TEXTLIST CmdTxtList
  0 = 'INITIALISE'
  1 = 'AlarmReset'
  2 = 'ColumnAlarmReset'
  3 = 'TIUSlideIn'
  4 = 'TIUSlideOut'
  5 = 'TIUDrawerUp'
  6 = 'TIUDrawerDown'
  7 = 'TIUSlideOutRetry'
  8 = 'TIUSlideOutCancel'
  9 = 'DPSPowerON'
  10 = 'DPSPowerOFF'
  11 = 'DPSPowerAuto'
  12 = 'AP240ACPowerON'
  13 = 'AP240ACPowerOFF'
  14 = 'APAirValveON'
  15 = 'APAirValveOFF'
  16 = 'TstAirValveON'
  17 = 'TstAirValveOFF'
  18 = 'CellDoorOpen'
  19 = 'CellDoorClose'
  20 = 'CancelBuffer'
  21 = 'SetLEDON'
  22 = 'SetLEDOFF'
  23 = 'SetLEDBlink'
  24 = 'DCCellFrontDoorOpen'
  25 = 'DCCellFrontDoorClose'
  26 = 'TIUSocketAirOn_1'
  27 = 'TIUSocketAirOn_2'
  28 = 'TIUSocketAirOff_1'
  29 = 'TIUSocketAirOff_2'
  30 = 'EnableTester'
  31 = 'DisableTester'
  32 = 'EnableTCU'
  33 = 'DisableTCU'
  34 = 'EnableTII'
  35 = 'DisableTII'
  36 = 'SetTCUSafeState'
  37 = 'SetSolenoidValvesON'
  38 = 'SetSolenoidValvesOFF'
  39 = 'Secondary24VPowerON'
  40 = 'Secondary24VPowerOFF'
   = ''
END_TEXTLIST

(* stored: Version 1.1.0.1, ProductVersion 3.1.4022.18
   TextList CmdTxtList: Id {223462ef-10ac-46cc-9510-ac4ce53d0ec0} *)
